_w1 := (gvl.BCV[BCV_Mapping.BCV_Caustic_Return].Status=Burkert.eBCV_Status.A_Closed) OR (gvl.BCV[BCV_Mapping.BCV_Caustic_Return].Status=Burkert.eBCV_Status.LOCKED_OUT);
_w2 := (gvl.BCV[BCV_Mapping.BCV_acid_Return].Status=Burkert.eBCV_Status.A_Closed) OR (gvl.BCV[BCV_Mapping.BCV_acid_Return].Status=Burkert.eBCV_Status.LOCKED_OUT);
_w3 := (gvl.BCV[BCV_Mapping.BCV_Caustic_Supply].Status=Burkert.eBCV_Status.A_Closed) OR (gvl.BCV[BCV_Mapping.BCV_Caustic_Supply].Status=Burkert.eBCV_Status.LOCKED_OUT);
_w4 := (gvl.BCV[BCV_Mapping.BCV_Acid_Supply].Status=Burkert.eBCV_Status.A_Closed) OR (gvl.BCV[BCV_Mapping.BCV_Acid_Supply].Status=Burkert.eBCV_Status.LOCKED_OUT);
_w5 := (Config.CIP_CTRL.Status=eCip_Status.Fill_Acid) AND _w1 AND _w3 OR (Config.CIP_CTRL.Status=eCip_Status.Fill_Rinse) AND (gvl.BCV[BCV_Mapping.BCV_Caustic_Return].Status=Burkert.eBCV_Status.A_Closed) AND (gvl.BCV[BCV_Mapping.BCV_Caustic_Supply].Status=Burkert.eBCV_Status.A_Closed) OR (Config.CIP_CTRL.Status=eCip_Status.Fill_Caustic) AND _w2 AND _w4 OR (Config.CIP_CTRL.Status=eCip_Status.Heat_Acid) AND _w1 AND _w3 OR (Config.CIP_CTRL.Status=eCip_Status.Heat_Rinse) AND _w1 AND _w3 OR (Config.CIP_CTRL.Status=eCip_Status.Heat_Caustic) AND _w2 AND _w4 OR (Config.CIP_CTRL.Status=eCip_Status.Low_Acid) AND _w1 AND _w3 OR (Config.CIP_CTRL.Status=eCip_Status.Low_Caustic) AND _w2 AND _w4;
F_TRIG_0(CLK := _w5); // F_trig
TON_1(IN := _w5, PT := T#1s); // TON
R_TRIG_0(CLK := TON_1.Q); // R_trig
PVL.PID[PID_Mapping.CIP_Supply_PID].PLC_Enable := SEL(F_TRIG_0.Q, SEL(R_TRIG_0.Q, PVL.PID[PID_Mapping.CIP_Supply_PID].PLC_Enable, True), False);
IF _w5 THEN _w6 := 50; END_IF
PVL.PID[PID_Mapping.CIP_Supply_PID].PLC_Target := _w6;
GVL.Vacon_VFD[Vacon_VFD_Mapping.CIP_Discharge].CONTROL.PLC_Run := PVL.PID[PID_Mapping.CIP_Supply_PID].PLC_Enable OR (PVL.PID[PID_Mapping.CIP_Supply_PID].MODE=ePID_Modes.FORCED_ON);
_w7 := Sanitizer_Target_Rate <> 0;
_w8 := Config.CIP_CTRL.Sanitzer_pump_LPM / 60;
// 253 ml /s
Sanitize_LPS := _w8;
_w9 := _w8 * Sanitize_Min_Pump_Time;
// 1.26 L for 5 Second Pump
Sanitizer_Min_Volume := _w9;
_w10 := (PVL.FIT[FIT_Mapping.CIP_Supply_Flow].Rate/60) * Config.CIP_CTRL.Sanizer_VPL;
Sanitizer_Target_Rate := _w10;
IF _w7 THEN _w11 := _w9 / _w10; END_IF
Santizer_Rest_Time := _w11 - Sanitize_Min_Pump_Time;
_w12 := (Config.CIP_CTRL.Status=eCIP_Status.Sanitize) AND (PVL.FIT[FIT_Mapping.CIP_Supply_Flow].Rate>10);
R_TRIG_2(CLK := _w12); // R_trig
_w13 := SEL(R_TRIG_2.Q, Santizer_Dispense_Volume, 0.0);
TON_0(IN := _w12, PT := T#2s); // TON
TP_1(IN := TON_0.Q AND NOT TP_2.Q, PT := REAL_TO_TIME(Sanitize_Min_Pump_Time) * 1000); // TP
gvl.BCV[bcv_mapping.BCV_Sanitizer_Inject].PLC_CMD := TP_1.Q;
F_TRIG_2(CLK := TP_1.Q); // F_Trig
Santizer_Dispense_Volume := SEL(F_TRIG_2.Q, _w13, Santizer_Dispense_Volume+Sanitizer_Min_Volume);
_w14 := PVL.CIP_Target[Config.CIP_CTRL.Target].Sanitize_Volume * Config.CIP_CTRL.Sanizer_VPL;
Sanitizer_Target_Volume := _w14;
_w15 := _w14 / Sanitize_LPS;
Santizer_Total_Time := _w15;
_w16 := Sanitize_Duration / (_w15 / Sanitize_Min_Pump_Time) - Sanitize_Min_Pump_Time;
Pump_OFF_Time := _w16;
TP_2(IN := F_TRIG_2.Q, PT := REAL_TO_TIME(_w16 * 1000)); // TP
IF (PVL.FIT[FIT_Mapping.CIP_Supply_Flow].Rate/60) <> 0 THEN _w17 := PVL.CIP_Target[Config.CIP_CTRL.Target].Sanitize_Volume / (PVL.FIT[FIT_Mapping.CIP_Supply_Flow].Rate/60); END_IF
Sanitize_Duration := _w17;
GVL.BCV[BCV_Mapping.BCV_Acid_Inject].PLC_CMD := ((Config.CIP_CTRL.Status=eCIP_Status.Low_Acid) OR (Config.CIP_CTRL.Status=eCIP_Status.Heat_Acid)) AND ((PVL.AIT[AIT_MApping.CIP_Acid_CND].Status=AIT_Status.Low_Low_Alarm) OR (PVL.AIT[AIT_MApping.CIP_Acid_CND].Status=AIT_Status.Low_Warning));
(* PVL.AIT[AIT_MApping.CIP_Return_CND].EU < PVL.AIT[AIT_MApping.CIP_Acid_CND].Burkert.cAlarm_Config.Low_warn; result not used *)
GVL.BCV[BCV_Mapping.BCV_Caustic_Inject].PLC_CMD := ((Config.CIP_CTRL.Status=eCIP_Status.Low_Caustic) OR (Config.CIP_CTRL.Status=eCIP_Status.Heat_Caustic)) AND ((PVL.AIT[AIT_MApping.CIP_Caustic_CND].Status=AIT_Status.Low_Low_Alarm) OR (PVL.AIT[AIT_MApping.CIP_Caustic_CND].Status=AIT_Status.Low_Warning));
(* PVL.AIT[AIT_MApping.CIP_Return_CND].EU < PVL.AIT[AIT_MApping.CIP_Caustic_CND].Burkert.cAlarm_Config.Low_warn; result not used *)
// Santizer_Rest_Time: input not connected

END_PROGRAM

// Alarms
ACTION Alarms:
ALARM_2_1(
    X := FloWave.Temp,
    LO_1 := floWave.Burkert.cAlarm_Config[1].Low_warn,
    HI_1 := floWave.Burkert.cAlarm_Config[1].Hi_Warn,
    LO_2 := floWave.Burkert.cAlarm_Config[1].Low_Low_Alarm,
    HI_2 := floWave.Burkert.cAlarm_Config[1].Hi_Hi_Alarm,
    HYS := 0.5); // BURKERT_OSCAT_BASIC.ALARM_2
ALARM_2_3(
    X := FloWave.Density_Factor,
    LO_1 := floWave.Burkert.cAlarm_Config[2].Low_warn,
    HI_1 := floWave.Burkert.cAlarm_Config[2].Hi_Warn,
    LO_2 := floWave.Burkert.cAlarm_Config[2].Low_Low_Alarm,
    HI_2 := floWave.Burkert.cAlarm_Config[2].Hi_Hi_Alarm,
    HYS := 0.5); // BURKERT_OSCAT_BASIC.ALARM_2
ALARM_2_0(
    X := FloWave.Concentration_2,
    LO_1 := floWave.Burkert.cAlarm_Config[0].Low_warn,
    HI_1 := floWave.Burkert.cAlarm_Config[0].Hi_Warn,
    LO_2 := floWave.Burkert.cAlarm_Config[0].Low_Low_Alarm,
    HI_2 := floWave.Burkert.cAlarm_Config[0].Hi_Hi_Alarm,
    HYS := 0.1); // BURKERT_OSCAT_BASIC.ALARM_2
ALARM_2_0(
    X := FloWave.Concentration_1,
    LO_1 := floWave.Burkert.cAlarm_Config[0].Low_warn,
    HI_1 := floWave.Burkert.cAlarm_Config[0].Hi_Warn,
    LO_2 := floWave.Burkert.cAlarm_Config[0].Low_Low_Alarm,
    HI_2 := floWave.Burkert.cAlarm_Config[0].Hi_Hi_Alarm,
    HYS := 0.1); // BURKERT_OSCAT_BASIC.ALARM_2
FloWave.Status := SEL(ALARM_2_0.Q2_HI OR ALARM_2_1.Q2_HI OR ALARM_2_3.Q2_HI OR ALARM_2_0.Q2_HI, SEL(ALARM_2_0.Q1_HI OR ALARM_2_1.Q1_HI OR ALARM_2_3.Q1_HI OR ALARM_2_0.Q1_HI, SEL(ALARM_2_0.Q2_LO OR ALARM_2_1.Q2_LO OR ALARM_2_3.Q2_LO OR ALARM_2_0.Q2_LO, SEL(ALARM_2_0.Q1_LO OR ALARM_2_1.Q1_LO OR ALARM_2_3.Q1_LO OR ALARM_2_0.Q1_LO, eFloWave_Status.OK, eFloWave_Status.Low_Warning), eFloWave_Status.Low_Low_Alarm), eFloWave_Status.High_Warning), eFloWave_Status.High_High_Alarm);
END_ACTION
